Fanuc KAREL source: kc00027.KL

-- PROVISIONAL review KL for V1013-1; original PC SHA256 41aaff30622a3d3177eefeb1d69b35ce930f76d32695979d6e5619975dd4f777
-- Incomplete behavior may be omitted. Consult companion uncertainty JSON. Do not deploy.
PROGRAM KC00027
%NOLOCKGROUP
BEGIN
  -- UNRESOLVED_PC offsets 5-81; opcodes 27,22,1C,22,1C,22,1C,22,22,1C,22,22,22,31
  -- UNRESOLVED_PC offsets 86-90; opcodes 7F
END KC00027
